	// VFD (Variable Frequency Drive) and other variables
	_0303_05_1_ixSection1_OverheatAlarm : BOOL;
	_0303_05_1_ixSection1_OverheatWarning : BOOL;
	_0303_05_1_ixVFD_Failure : BOOL;
	_0303_05_1_ixVFD_InWork : BOOL;
	_0303_05_1_ixVFD_Manual : BOOL;
	_0303_05_1_ixVFD_Ready : BOOL;
	_0303_05_1KM8_ixStatusOn : BOOL;
	_0303_05_2_ixSection1_OverheatAlarm : BOOL;
	_0303_05_2_ixSection1_OverheatWarning : BOOL;
	_0303_05_2_ixVFD_Failure : BOOL;
	_0303_05_2_ixVFD_InWork : BOOL;
	_0303_05_2_ixVFD_Manual : BOOL;
	_0303_05_2_ixVFD_Ready : BOOL;
	_0303_05_2KM8_ixStatusOn : BOOL;
	
	// Выходы
	_0303_05_BY01_qxShutter_Open        : BOOL;
	_0303_05_BY01_qxShutter_Close       : BOOL;
	_0303_05_BY02_qxShutter_Open        : BOOL;
	_0303_05_BY02_qxShutter_Close       : BOOL;
	_0303_05_BY03_qxShutter_Open        : BOOL;
	_0303_05_BY03_qxShutter_Close       : BOOL;
	_0303_05_BY04_qxShutter_Open        : BOOL;
	_0303_05_BY04_qxShutter_Close       : BOOL;
	_0303_05_BY05_qxShutter_Open        : BOOL;
	_0303_05_BY05_qxShutter_Close       : BOOL;
	_0303_05_BY07_qxShutter_Open        : BOOL;
	_0303_05_BY07_qxShutter_Close       : BOOL;
	_0303_05_BY08_qxShutter_Open        : BOOL;
	_0303_05_BY08_qxShutter_Close       : BOOL;
	
	_0303_05_PU01_qxKM_cmdOn            : BOOL;
	_0303_05_PU01_qxKM_Frq_cmdOn        : BOOL;
	_0303_05_PU02_qxKM_cmdOn            : BOOL;
	_0303_05_PU02_qxKM_Frq_cmdOn        : BOOL;
	_0303_05_PU03_qxKM_cmdOn            : BOOL;
	_0303_05_PU03_qxKM_Frq_cmdOn        : BOOL;
	_0303_05_PU04_qxKM_cmdOn            : BOOL;
	_0303_05_PU04_qxKM_Frq_cmdOn        : BOOL;
	_0303_05_PU05_qxKM_cmdOn            : BOOL;
	_0303_05_PU05_qxKM_Frq_cmdOn		: BOOL;
	
	_0303_05_qxEmergencyStop : BOOL;			// Реле аварийного останова
	_0303_05_1KM8_qxOn : BOOL;					// Включить 1KM8
	_0303_05_2KM8_qxOn : BOOL;					// Включить 2KM8
	
	_0303_05_VFD001_qIMainFrq_SetFrq		: REAL;
	_0303_05_VFD002_qIReserveFrq_SetFrq		: REAL;
END_VAR
    TASK MainTask(INTERVAL := T#150ms, PRIORITY := 1);
    TASK VISU_TASK(INTERVAL := T#100ms, PRIORITY := 31);
    TASK SoftMotion_PlanningTask(INTERVAL := T#2ms, PRIORITY := 15);
    PROGRAM NEW_MAIN WITH MainTask : NEW_MAIN;
    PROGRAM VisuElems.Visu_Prg WITH VISU_TASK : VisuElems.Visu_Prg;
  END_RESOURCE
END_CONFIGURATION

CONFIGURATION Ethernet_1
END_CONFIGURATION

CONFIGURATION ModbusTCP_Slave_Device_1
END_CONFIGURATION

CONFIGURATION Modbus_TCP_Master_1
END_CONFIGURATION

CONFIGURATION MV210_202_1A3
END_CONFIGURATION

CONFIGURATION MV210_202_1A4
END_CONFIGURATION

CONFIGURATION MV210_202_1A5
END_CONFIGURATION

CONFIGURATION MU210_403_1A6
END_CONFIGURATION

CONFIGURATION MV210_101_1A7
END_CONFIGURATION

CONFIGURATION MU210_502_1A8
END_CONFIGURATION

CONFIGURATION MV210_202_1A2
END_CONFIGURATION

CONFIGURATION Modbus_COM
END_CONFIGURATION

CONFIGURATION Modbus_Master_COM_Port
END_CONFIGURATION

CONFIGURATION TKC1
END_CONFIGURATION

CONFIGURATION TKC2
END_CONFIGURATION

CONFIGURATION _1UZ8
END_CONFIGURATION

CONFIGURATION _2UZ8
END_CONFIGURATION

CONFIGURATION Modbus_COM_1
END_CONFIGURATION

CONFIGURATION Modbus_Master_COM_Port_1
END_CONFIGURATION

CONFIGURATION MBSlave_ZRA_1
END_CONFIGURATION

CONFIGURATION MBSlave_ZRA_2
END_CONFIGURATION

CONFIGURATION MBSlave_ZRA_3
END_CONFIGURATION

CONFIGURATION MBSlave_ZRA_4
END_CONFIGURATION

CONFIGURATION MBSlave_ZRA_5
END_CONFIGURATION

CONFIGURATION MBSlave_ZRA_7
END_CONFIGURATION

CONFIGURATION MBSlave_ZRA_8
END_CONFIGURATION
